TYPE ST_CFG_STI_EtherCAT_Conveyor :
(**************************************************************************************
 * 	Application		:	BoxControl Framework
 *	Revision		:	$Revision: 354744 $
 *	Revision date	:	$Date: 2015-09-10 22:43:15 +0200 (Do, 10 Sep 2015) $
 *	Last changed by	:	$Author: d7mangc $
 *	URL				:	$URL: http://almscdc.swisslog.com/repo/SWPD/Development/BoxControlFramework/20_Release/trunk/01_Software/BoxControlFramework/BoxControlFramework/JumpStart/11_Library/10_Application/12_ElementFunctions/01_DUTs/ST_HW_InputsDummyFunction.TcDUT $
 *
 *	Purpose			:	Specific configuration for a conveyor Subsystem transport interface over EtherCAT
 *
 * ------------------------------------------------------------------------------------
 *	Copyright Swisslog [IP AG], Switzerland. All rights reserved.
 * 
 * ------------------------------------------------------------------------------------
 *	
 * 	Revision History: 
 *
 * 	VERSION			DATE			INITIALS			DESCRIPTION
 *	0.1				01.01.2001		swl					Example
 *
 **************************************************************************************)	
STRUCT
	eExternalFunctionNumber	: E_FunctionNumber; // Function number
	AdjFunctionNumber		: ST_PositionIdent; // Internal adjacent position
	Inbound					: BOOL; // Is inbound interface - FALSE = Outbound
	DeleteTU_Data			: BOOL := TRUE; // Inbound: Clears existing TU data slot which corresponds to data provided by the interface, Outbound: Deletes TU in own system after handover
	tWatchdog				: TIME; // Monitor communicaiton
	tHeartBeat				: TIME; // Time for generating watchdog heart beat
	OnlyFastSpeed			: BOOL; // Enable means FastSpeed always active, Disable = Controlled by interface
	OverwriteTU_Data		: BOOL := TRUE ; // TRUE = Overwrite existing TU data in the system with data from the interface, FALSE = Use interface data for identifiation only
END_STRUCT
END_TYPE

(* stored: Version 1.1.0.1, ProductVersion 3.1.4022.18
   DUT ST_CFG_STI_EtherCAT_Conveyor: Id {c2508dda-726a-4b1c-83ce-8a7dff9685a0} *)
